// TIA Portal project "Pompe" (V15.1)

(* hardware
DEVICE "S71500/ET200MP station_1"  S7-1500 station
   slot 0: "Rail_0"  Rack  6ES7 590-1***0-0AA0
   slot 1: "PLC_1"  CPU 1513-1 PN  6ES7 513-1AL02-0AB0  V2.6
      slot 3: "CPU display_1"  6ES7591-1AA00-0AA0
DEVICE "HMI_1"  KTP900 Basic PN
   slot 0: "HMI_1"  KTP900 Basic PN  6AV2 123-2JB03-0AX0  15.1.0.0
   slot 1: "HMI_RT_1"  KTP900 Basic PN  6AV2 123-2JB03-0AX0  15.1.0.0
   slot 5: "HMI_1.IE_CP_1"  PROFINET Interface  15.0.1.0
      slot 1: "PROFINET Interface_1"  PROFINET Interface
         slot 1: "Port_1"  Port
*)

// ===== PLC "PLC_1"  CPU 1513-1 PN =====

VAR_GLOBAL   // PLC tag table "Default tag table"
   "Clock_Byte" AT %MB0 : Byte;
   "Clock_10Hz" AT %M0.0 : Bool;
   "Clock_5Hz" AT %M0.1 : Bool;
   "Clock_2.5Hz" AT %M0.2 : Bool;
   "Clock_2Hz" AT %M0.3 : Bool;
   "Clock_1.25Hz" AT %M0.4 : Bool;
   "Clock_1Hz" AT %M0.5 : Bool;
   "Clock_0.625Hz" AT %M0.6 : Bool;
   "Clock_0.5Hz" AT %M0.7 : Bool;
END_VAR

DATA_BLOCK "Pompa_DB"   // DB1
{ S7_Optimized_Access := 'TRUE' }
VERSION : 0.1
   VAR
      comanda_start : Bool;
      comanda_oprire : Bool;
      feedback : Bool;
      pornire_succes : Bool;
   END_VAR
BEGIN
END_DATA_BLOCK

DATA_BLOCK "Bazin_DB"   // DB2
{ S7_Optimized_Access := 'TRUE' }
VERSION : 0.1
   VAR
      volum_maxim : Real := 100.0;
      volum_curent : Real;
      gol : Bool;
      plin : Bool;
   END_VAR
BEGIN
END_DATA_BLOCK

DATA_BLOCK "Robinet_DB"   // DB3
{ S7_Optimized_Access := 'TRUE' }
VERSION : 0.1
   VAR
      comanda_pornire : Bool;
      pornit : Bool;
      comanda_oprire : Bool;
   END_VAR
BEGIN
END_DATA_BLOCK

DATA_BLOCK "Alarme"   // DB4
{ S7_Optimized_Access := 'TRUE' }
VERSION : 0.1
   VAR
      alarme_gather : Word;
      alarme_vect : Array[0..15] of Bool;
   END_VAR
BEGIN
END_DATA_BLOCK

DATA_BLOCK "Avarii"   // DB5
{ S7_Optimized_Access := 'TRUE' }
VERSION : 0.1
   VAR
      esd : Bool;
      btn_esd : Bool;
      btn_reset_esd : Bool;
      avarie_pompa_1 : Bool;
      avarie_pompa_auxiliara : Bool;
      avarie_robinet : Bool;
      avarie_generala : Bool;
      reset_avarie_generala : Bool;
   END_VAR
BEGIN
END_DATA_BLOCK

DATA_BLOCK "Butoane/Permisiuni"   // DB6
{ S7_Optimized_Access := 'TRUE' }
VERSION : 0.1
BEGIN
END_DATA_BLOCK

DATA_BLOCK "Simulare_DB"   // DB9
{ S7_Optimized_Access := 'TRUE' }
VERSION : 0.1
   VAR
      mod_selectat : USInt;
      paritate_mod : USInt;
      pompa_oprita_hmi : Bool;
      pompa_aux_oprita_hmi : Bool;
      robinet_oprit_hmi : Bool;
      nivel_de_mentinut : Real;
   END_VAR
BEGIN
END_DATA_BLOCK

DATA_BLOCK "Bazin_DB_1"   // DB10
{ S7_Optimized_Access := 'TRUE' }
VERSION : 0.1
// stored: InstanceOfName Bazin
"Bazin"
BEGIN
END_DATA_BLOCK

DATA_BLOCK "Robinet_DB_1"   // DB11
{ S7_Optimized_Access := 'TRUE' }
VERSION : 0.1
// stored: InstanceOfName Robinet
"Robinet"
BEGIN
END_DATA_BLOCK

DATA_BLOCK "Auxiliare"   // DB12
{ S7_Optimized_Access := 'TRUE' }
VERSION : 0.1
   VAR
      enable_network : Bool := false;
   END_VAR
BEGIN
END_DATA_BLOCK

DATA_BLOCK "Vana_DB"   // DB13
{ S7_Optimized_Access := 'TRUE' }
VERSION : 0.1
   VAR
      comanda_start : Bool;
      comanda_oprire : Bool;
      feedback : Bool;
      pornire_succes : Bool;
   END_VAR
BEGIN
END_DATA_BLOCK

DATA_BLOCK "Vana_DB_1"   // DB14
{ S7_Optimized_Access := 'TRUE' }
VERSION : 0.1
// stored: InstanceOfName Vana
"Vana"
BEGIN
END_DATA_BLOCK

DATA_BLOCK "Pompa_DB_1"   // DB15
{ S7_Optimized_Access := 'TRUE' }
VERSION : 0.1
// stored: InstanceOfName Pompa
"Pompa"
BEGIN
END_DATA_BLOCK

DATA_BLOCK "Simulare_DB_1"   // DB16
{ S7_Optimized_Access := 'TRUE' }
VERSION : 0.1
// stored: InstanceOfName Simulare
"Simulare"
BEGIN
END_DATA_BLOCK

DATA_BLOCK "Pompa_DB_2"   // DB17
{ S7_Optimized_Access := 'TRUE' }
VERSION : 0.1
// stored: InstanceOfName Pompa
"Pompa"
BEGIN
END_DATA_BLOCK

DATA_BLOCK "Pompa_auxiliara_DB"   // DB18
{ S7_Optimized_Access := 'TRUE' }
VERSION : 0.1
   VAR
      comanda_start : Bool;
      comanda_oprire : Bool;
      feedback : Bool;
      pornire_succes : Bool;
      btn_pornire : Bool;
   END_VAR
BEGIN
END_DATA_BLOCK

// folder: System blocks/Program resources

DATA_BLOCK "Timer_reset_ESD"   // DB7
{ S7_Optimized_Access := 'TRUE' }
AUTHOR : Simatic
FAMILY : IEC
NAME : IEC_TMR
VERSION : 1.0
// stored: InstanceOfName IEC_TIMER
"IEC_TIMER"
BEGIN
END_DATA_BLOCK

DATA_BLOCK "Timer_reset_avarie_generala"   // DB8
{ S7_Optimized_Access := 'TRUE' }
AUTHOR : Simatic
FAMILY : IEC
NAME : IEC_TMR
VERSION : 1.0
// stored: InstanceOfName IEC_TIMER
"IEC_TIMER"
BEGIN
END_DATA_BLOCK

// folder: (top level)

FUNCTION_BLOCK "Pompa"   // FB1, LAD
{ S7_Optimized_Access := 'TRUE' }
VERSION : 0.1
   VAR_INPUT
      esd : Bool;
      avarie : Bool;
      mod_selectat : USInt;
      comanda_oprire : Bool;
   END_VAR
   VAR_OUTPUT
      feedback : Bool;
      pornire_succes : Bool;
   END_VAR
   VAR_IN_OUT
      comanda_start : Bool;
   END_VAR
   VAR
      pornire : Bool;
      timer_confirmare : TON_TIME;
   END_VAR
BEGIN

REGION Network 1: Comanda plecare
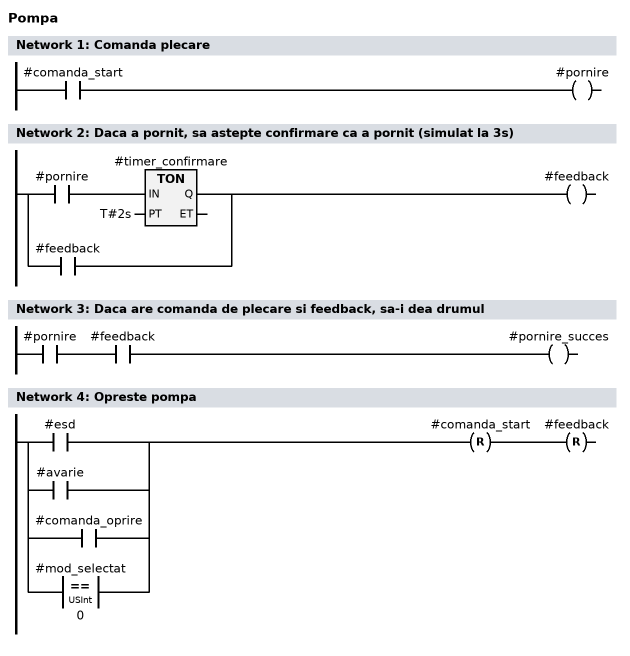
   RUNG wire#powerrail
      Contact( #comanda_start )
      Coil( #pornire )
   END_RUNG
   // the same network as SCL:
   #pornire := #comanda_start;
END_REGION

REGION Network 2: Daca a pornit, sa astepte confirmare ca a pornit (simulat la 3s)
   #timer_confirmare(IN := #pornire, PT := T#2s);   // TON
   #feedback := #timer_confirmare.Q OR #feedback;
END_REGION

REGION Network 3: Daca are comanda de plecare si feedback, sa-i dea drumul
   RUNG wire#powerrail
      Contact( #pornire )
      Contact( #feedback )
      Coil( #pornire_succes )
   END_RUNG
   // the same network as SCL:
   #pornire_succes := #pornire AND #feedback;
END_REGION

REGION Network 4: Opreste pompa
   RUNG wire#powerrail
      Contact( #esd )
      wire#w1
      R_Coil( #comanda_start )
      R_Coil( #feedback )
   END_RUNG
   RUNG wire#powerrail
      Contact( #avarie )
   END_RUNG wire#w1
   RUNG wire#powerrail
      Contact( #comanda_oprire )
   END_RUNG wire#w1
   RUNG wire#powerrail
      { S7_Templates := "SrcType := USInt" } EQ_Contact(in1 := #mod_selectat, in2 := 0)
   END_RUNG wire#w1
   // the same network as SCL:
   IF #esd OR #avarie OR #comanda_oprire OR (#mod_selectat = 0) THEN
       #comanda_start := FALSE;
       #feedback := FALSE;
   END_IF;
END_REGION
END_FUNCTION_BLOCK

FUNCTION_BLOCK "Bazin"   // FB2, LAD
{ S7_Optimized_Access := 'TRUE' }
VERSION : 0.1
   VAR_INPUT
      volum_maxim : Real;
   END_VAR
   VAR_OUTPUT
      gol : Bool;
      plin : Bool;
   END_VAR
   VAR_IN_OUT
      volum_curent : Real;
   END_VAR
BEGIN

REGION Network 1: Setare gol
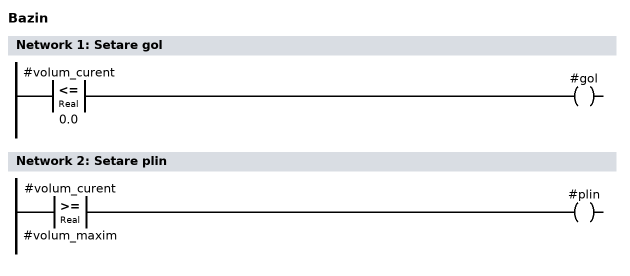
   RUNG wire#powerrail
      { S7_Templates := "SrcType := Real" } LE_Contact(in1 := #volum_curent, in2 := 0.0)
      Coil( #gol )
   END_RUNG
   // the same network as SCL:
   #gol := #volum_curent <= 0.0;
END_REGION

REGION Network 2: Setare plin
   RUNG wire#powerrail
      { S7_Templates := "SrcType := Real" } GE_Contact(in1 := #volum_curent, in2 := #volum_maxim)
      Coil( #plin )
   END_RUNG
   // the same network as SCL:
   #plin := #volum_curent >= #volum_maxim;
END_REGION
END_FUNCTION_BLOCK

FUNCTION_BLOCK "Robinet"   // FB3, LAD
{ S7_Optimized_Access := 'TRUE' }
VERSION : 0.1
   VAR_INPUT
      esd : Bool;
      avarie : Bool;
      comanda_oprire : Bool;
   END_VAR
   VAR_IN_OUT
      pornit : Bool;
      btn_pornire : Bool;
   END_VAR
BEGIN

REGION Network 1: Sa aiba permisiunea de pornire
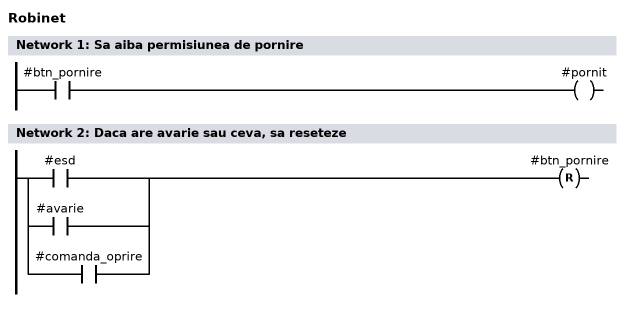
   RUNG wire#powerrail
      Contact( #btn_pornire )
      Coil( #pornit )
   END_RUNG
   // the same network as SCL:
   #pornit := #btn_pornire;
END_REGION

REGION Network 2: Daca are avarie sau ceva, sa reseteze
   RUNG wire#powerrail
      Contact( #esd )
      wire#w1
      R_Coil( #btn_pornire )
   END_RUNG
   RUNG wire#powerrail
      Contact( #avarie )
   END_RUNG wire#w1
   RUNG wire#powerrail
      Contact( #comanda_oprire )
   END_RUNG wire#w1
   // the same network as SCL:
   IF #esd OR #avarie OR #comanda_oprire THEN #btn_pornire := FALSE; END_IF;
END_REGION
END_FUNCTION_BLOCK

FUNCTION_BLOCK "Simulare"   // FB4, LAD
{ S7_Optimized_Access := 'TRUE' }
VERSION : 0.1
   VAR_INPUT
      plin : Bool;
      gol : Bool;
      pompa_pornita : Bool;
      pompa_aux_pornita : Bool;
      robinet_pornit : Bool;
      esd : Bool;
      avarie_pompa : Bool;
      avarie_pompa_aux : Bool;
      avarie_robinet : Bool;
      nivel_de_mentinut : Real;
   END_VAR
   VAR_OUTPUT
      start_pompa : Bool;
      start_pompa_aux : Bool;
      start_robinet : Bool;
      opreste_pompa : Bool;
      opreste_pompa_aux : Bool;
      opreste_robinet : Bool;
      pompa_oprita_hmi : Bool;
      pompa_oprita_aux_hmi : Bool;
      robinet_oprit_hmi : Bool;
   END_VAR
   VAR_IN_OUT
      btn_pompa_aux : Bool;
      volum_curent : Real;
      mod_functionare : USInt;
   END_VAR
   VAR
      re1 : Bool;
      re2 : Bool;
      re3 : Bool;
      lim_inf : Real;
      lim_sup : Real;
   END_VAR
   VAR_TEMP   // added for the SCL form of the ladder/FBD networks
      _w1 : Bool;
      _w2 : Bool;
   END_VAR
BEGIN

REGION Network 1: Calcul limite noi
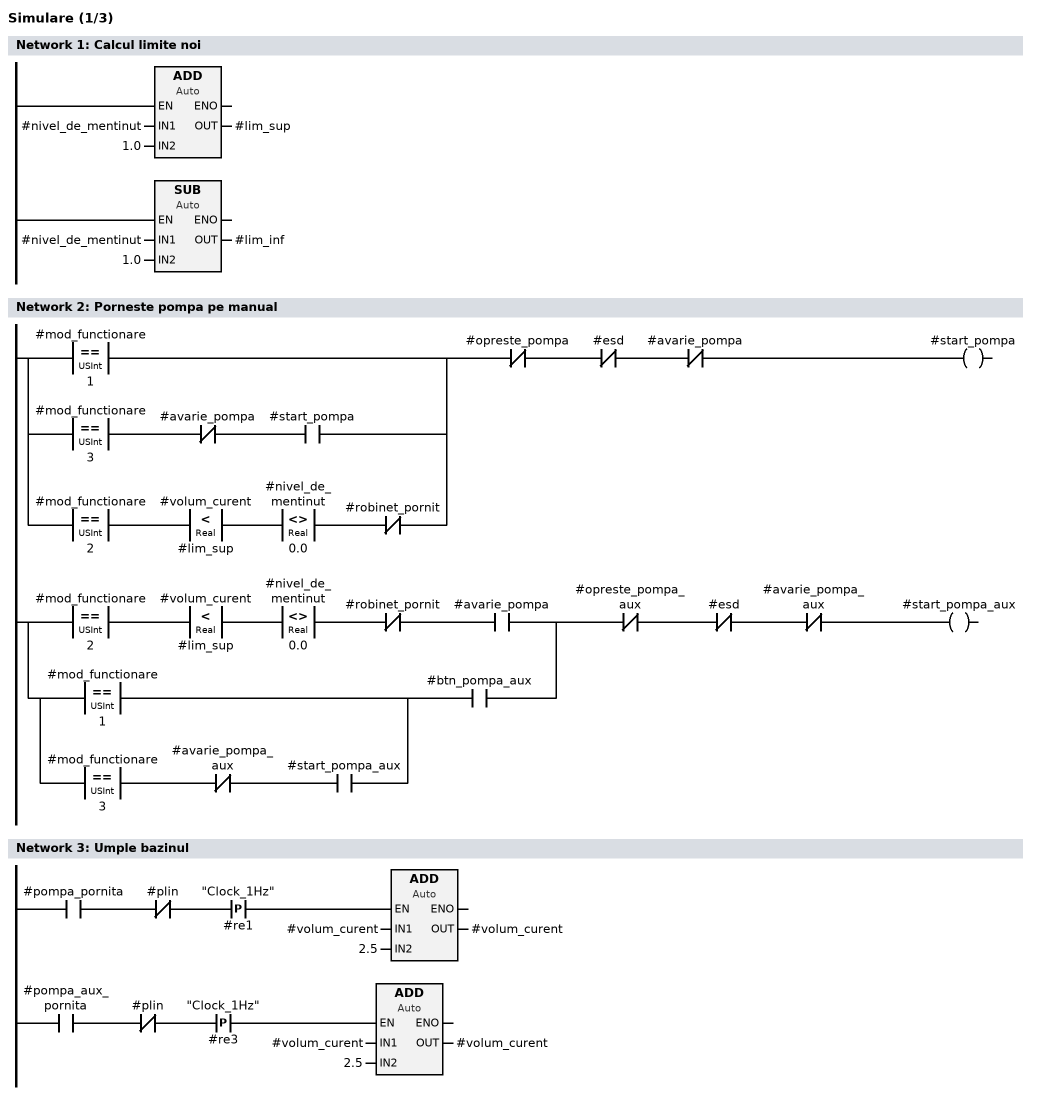
   RUNG wire#powerrail
      Add(in1 := #nivel_de_mentinut, in2 := 1.0, out => #lim_sup)
   END_RUNG
   RUNG wire#powerrail
      Sub(in1 := #nivel_de_mentinut, in2 := 1.0, out => #lim_inf)
   END_RUNG
   // the same network as SCL:
   #lim_sup := #nivel_de_mentinut + 1.0;
   #lim_inf := #nivel_de_mentinut - 1.0;
END_REGION

REGION Network 2: Porneste pompa pe manual
   RUNG wire#powerrail
      { S7_Templates := "SrcType := USInt" } EQ_Contact(in1 := #mod_functionare, in2 := 1)
      wire#w1
      I_Contact( #opreste_pompa )
      I_Contact( #esd )
      I_Contact( #avarie_pompa )
      Coil( #start_pompa )
   END_RUNG
   RUNG wire#powerrail
      { S7_Templates := "SrcType := USInt" } EQ_Contact(in1 := #mod_functionare, in2 := 3)
      I_Contact( #avarie_pompa )
      Contact( #start_pompa )
   END_RUNG wire#w1
   RUNG wire#powerrail
      { S7_Templates := "SrcType := USInt" } EQ_Contact(in1 := #mod_functionare, in2 := 2)
      { S7_Templates := "SrcType := Real" } LT_Contact(in1 := #volum_curent, in2 := #lim_sup)
      { S7_Templates := "SrcType := Real" } NE_Contact(in1 := #nivel_de_mentinut, in2 := 0.0)
      I_Contact( #robinet_pornit )
   END_RUNG wire#w1
   RUNG wire#powerrail
      { S7_Templates := "SrcType := USInt" } EQ_Contact(in1 := #mod_functionare, in2 := 2)
      { S7_Templates := "SrcType := Real" } LT_Contact(in1 := #volum_curent, in2 := #lim_sup)
      { S7_Templates := "SrcType := Real" } NE_Contact(in1 := #nivel_de_mentinut, in2 := 0.0)
      I_Contact( #robinet_pornit )
      Contact( #avarie_pompa )
      wire#w2
      I_Contact( #opreste_pompa_aux )
      I_Contact( #esd )
      I_Contact( #avarie_pompa_aux )
      Coil( #start_pompa_aux )
   END_RUNG
   RUNG wire#powerrail
      { S7_Templates := "SrcType := USInt" } EQ_Contact(in1 := #mod_functionare, in2 := 1)
      wire#w3
      Contact( #btn_pompa_aux )
   END_RUNG wire#w2
   RUNG wire#powerrail
      { S7_Templates := "SrcType := USInt" } EQ_Contact(in1 := #mod_functionare, in2 := 3)
      I_Contact( #avarie_pompa_aux )
      Contact( #start_pompa_aux )
   END_RUNG wire#w3
   // the same network as SCL:
   #start_pompa := ((#mod_functionare = 1) OR ((#mod_functionare = 3) AND NOT #avarie_pompa AND #start_pompa) OR ((#mod_functionare = 2) AND (#volum_curent < #lim_sup) AND (#nivel_de_mentinut <> 0.0) AND NOT #robinet_pornit)) AND NOT #opreste_pompa AND NOT #esd AND NOT #avarie_pompa;
   #start_pompa_aux := (((#mod_functionare = 2) AND (#volum_curent < #lim_sup) AND (#nivel_de_mentinut <> 0.0) AND NOT #robinet_pornit AND #avarie_pompa) OR (((#mod_functionare = 1) OR ((#mod_functionare = 3) AND NOT #avarie_pompa_aux AND #start_pompa_aux)) AND #btn_pompa_aux)) AND NOT #opreste_pompa_aux AND NOT #esd AND NOT #avarie_pompa_aux;
END_REGION

REGION Network 3: Umple bazinul
   RUNG wire#powerrail
      Contact( #pompa_pornita )
      I_Contact( #plin )
      P_Contact(operand := "Clock_1Hz", bit := #re1)
      Add(in1 := #volum_curent, in2 := 2.5, out => #volum_curent)
   END_RUNG
   RUNG wire#powerrail
      Contact( #pompa_aux_pornita )
      I_Contact( #plin )
      P_Contact(operand := "Clock_1Hz", bit := #re3)
      Add(in1 := #volum_curent, in2 := 2.5, out => #volum_curent)
   END_RUNG
   // the same network as SCL:
   #_w1 := #pompa_pornita AND NOT #plin AND "Clock_1Hz" AND NOT #re1;   // rising edge of "Clock_1Hz"
   #re1 := "Clock_1Hz";
   IF #_w1 THEN #volum_curent := #volum_curent + 2.5; END_IF;
   #_w2 := #pompa_aux_pornita AND NOT #plin AND "Clock_1Hz" AND NOT #re3;   // rising edge of "Clock_1Hz"
   #re3 := "Clock_1Hz";
   IF #_w2 THEN #volum_curent := #volum_curent + 2.5; END_IF;
END_REGION

REGION Network 4: Opreste pompa/pompa aux
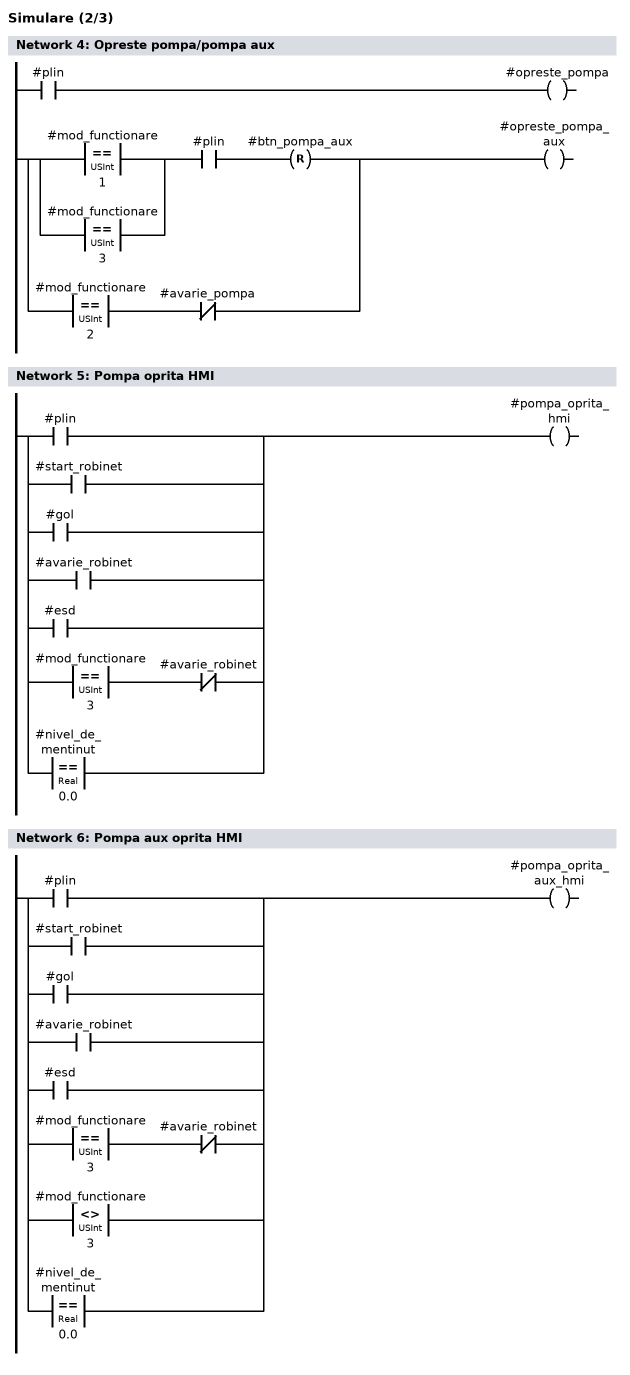
   RUNG wire#powerrail
      Contact( #plin )
      Coil( #opreste_pompa )
   END_RUNG
   RUNG wire#powerrail
      { S7_Templates := "SrcType := USInt" } EQ_Contact(in1 := #mod_functionare, in2 := 1)
      wire#w1
      Contact( #plin )
      R_Coil( #btn_pompa_aux )
      wire#w2
      Coil( #opreste_pompa_aux )
   END_RUNG
   RUNG wire#powerrail
      { S7_Templates := "SrcType := USInt" } EQ_Contact(in1 := #mod_functionare, in2 := 3)
   END_RUNG wire#w1
   RUNG wire#powerrail
      { S7_Templates := "SrcType := USInt" } EQ_Contact(in1 := #mod_functionare, in2 := 2)
      I_Contact( #avarie_pompa )
   END_RUNG wire#w2
   // the same network as SCL:
   #opreste_pompa := #plin;
   #_w1 := ((#mod_functionare = 1) OR (#mod_functionare = 3)) AND #plin;
   IF #_w1 THEN #btn_pompa_aux := FALSE; END_IF;
   #opreste_pompa_aux := #_w1 OR ((#mod_functionare = 2) AND NOT #avarie_pompa);
END_REGION

REGION Network 5: Pompa oprita HMI
   RUNG wire#powerrail
      Contact( #plin )
      wire#w1
      Coil( #pompa_oprita_hmi )
   END_RUNG
   RUNG wire#powerrail
      Contact( #start_robinet )
   END_RUNG wire#w1
   RUNG wire#powerrail
      Contact( #gol )
   END_RUNG wire#w1
   RUNG wire#powerrail
      Contact( #avarie_robinet )
   END_RUNG wire#w1
   RUNG wire#powerrail
      Contact( #esd )
   END_RUNG wire#w1
   RUNG wire#powerrail
      { S7_Templates := "SrcType := USInt" } EQ_Contact(in1 := #mod_functionare, in2 := 3)
      I_Contact( #avarie_robinet )
   END_RUNG wire#w1
   RUNG wire#powerrail
      { S7_Templates := "SrcType := Real" } EQ_Contact(in1 := #nivel_de_mentinut, in2 := 0.0)
   END_RUNG wire#w1
   // the same network as SCL:
   #pompa_oprita_hmi := #plin OR #start_robinet OR #gol OR #avarie_robinet OR #esd OR ((#mod_functionare = 3) AND NOT #avarie_robinet) OR (#nivel_de_mentinut = 0.0);
END_REGION

REGION Network 6: Pompa aux oprita HMI
   RUNG wire#powerrail
      Contact( #plin )
      wire#w1
      Coil( #pompa_oprita_aux_hmi )
   END_RUNG
   RUNG wire#powerrail
      Contact( #start_robinet )
   END_RUNG wire#w1
   RUNG wire#powerrail
      Contact( #gol )
   END_RUNG wire#w1
   RUNG wire#powerrail
      Contact( #avarie_robinet )
   END_RUNG wire#w1
   RUNG wire#powerrail
      Contact( #esd )
   END_RUNG wire#w1
   RUNG wire#powerrail
      { S7_Templates := "SrcType := USInt" } EQ_Contact(in1 := #mod_functionare, in2 := 3)
      I_Contact( #avarie_robinet )
   END_RUNG wire#w1
   RUNG wire#powerrail
      { S7_Templates := "SrcType := USInt" } NE_Contact(in1 := #mod_functionare, in2 := 3)
   END_RUNG wire#w1
   RUNG wire#powerrail
      { S7_Templates := "SrcType := Real" } EQ_Contact(in1 := #nivel_de_mentinut, in2 := 0.0)
   END_RUNG wire#w1
   // the same network as SCL:
   #pompa_oprita_aux_hmi := #plin OR #start_robinet OR #gol OR #avarie_robinet OR #esd OR ((#mod_functionare = 3) AND NOT #avarie_robinet) OR (#mod_functionare <> 3) OR (#nivel_de_mentinut = 0.0);
END_REGION

REGION Network 7: Robinet oprit HMI
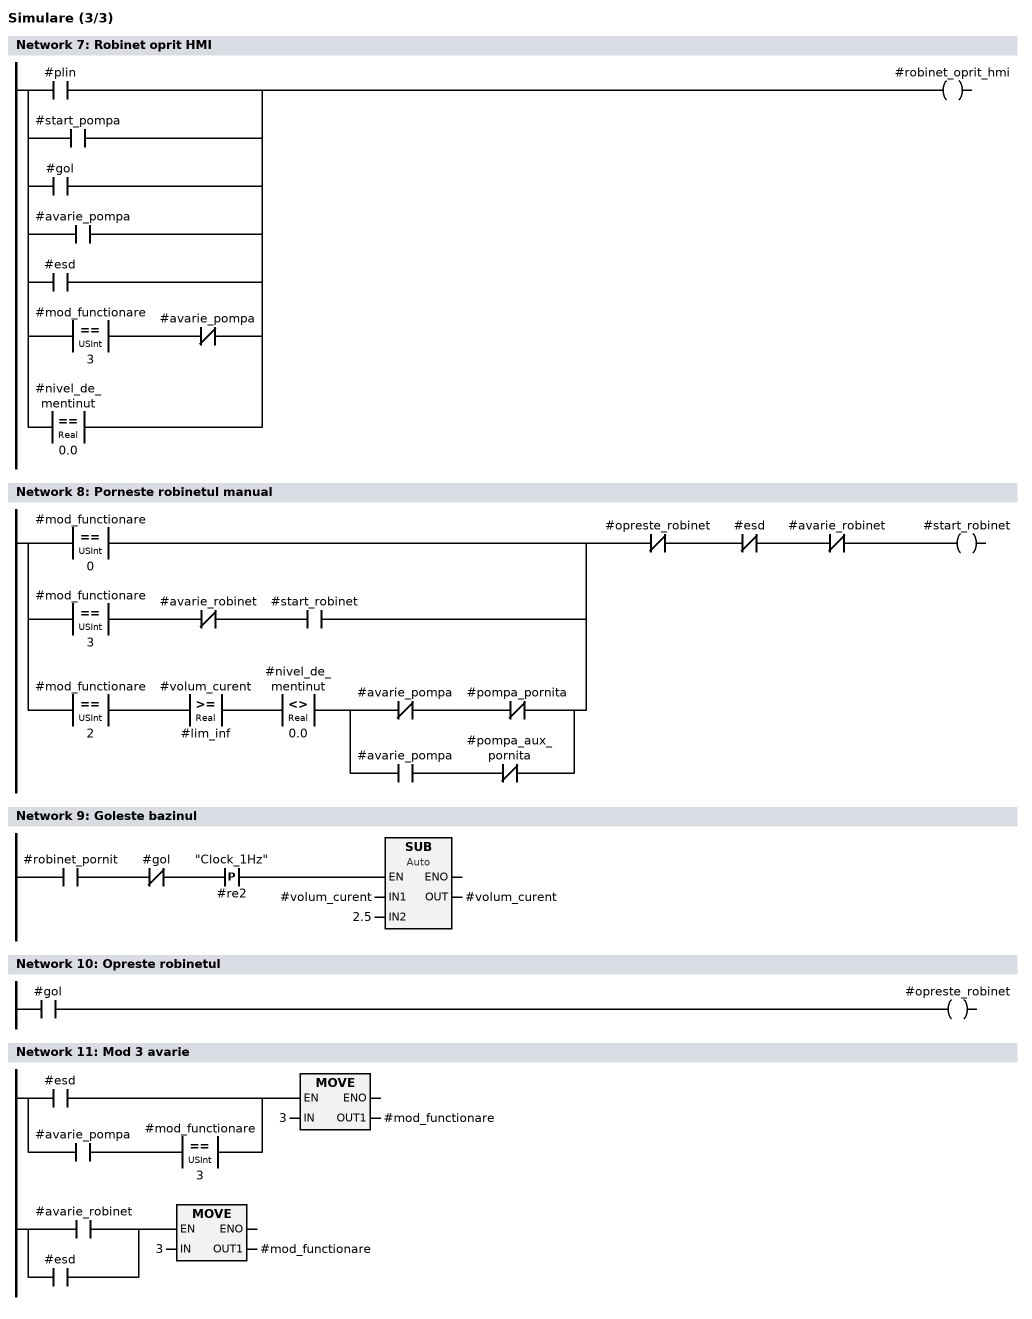
   RUNG wire#powerrail
      Contact( #plin )
      wire#w1
      Coil( #robinet_oprit_hmi )
   END_RUNG
   RUNG wire#powerrail
      Contact( #start_pompa )
   END_RUNG wire#w1
   RUNG wire#powerrail
      Contact( #gol )
   END_RUNG wire#w1
   RUNG wire#powerrail
      Contact( #avarie_pompa )
   END_RUNG wire#w1
   RUNG wire#powerrail
      Contact( #esd )
   END_RUNG wire#w1
   RUNG wire#powerrail
      { S7_Templates := "SrcType := USInt" } EQ_Contact(in1 := #mod_functionare, in2 := 3)
      I_Contact( #avarie_pompa )
   END_RUNG wire#w1
   RUNG wire#powerrail
      { S7_Templates := "SrcType := Real" } EQ_Contact(in1 := #nivel_de_mentinut, in2 := 0.0)
   END_RUNG wire#w1
   // the same network as SCL:
   #robinet_oprit_hmi := #plin OR #start_pompa OR #gol OR #avarie_pompa OR #esd OR ((#mod_functionare = 3) AND NOT #avarie_pompa) OR (#nivel_de_mentinut = 0.0);
END_REGION

REGION Network 8: Porneste robinetul manual
   RUNG wire#powerrail
      { S7_Templates := "SrcType := USInt" } EQ_Contact(in1 := #mod_functionare, in2 := 0)
      wire#w1
      I_Contact( #opreste_robinet )
      I_Contact( #esd )
      I_Contact( #avarie_robinet )
      Coil( #start_robinet )
   END_RUNG
   RUNG wire#powerrail
      { S7_Templates := "SrcType := USInt" } EQ_Contact(in1 := #mod_functionare, in2 := 3)
      I_Contact( #avarie_robinet )
      Contact( #start_robinet )
   END_RUNG wire#w1
   RUNG wire#powerrail
      { S7_Templates := "SrcType := USInt" } EQ_Contact(in1 := #mod_functionare, in2 := 2)
      { S7_Templates := "SrcType := Real" } GE_Contact(in1 := #volum_curent, in2 := #lim_inf)
      { S7_Templates := "SrcType := Real" } NE_Contact(in1 := #nivel_de_mentinut, in2 := 0.0)
      wire#w2
      I_Contact( #avarie_pompa )
      I_Contact( #pompa_pornita )
   END_RUNG wire#w1
   RUNG wire#w2
      Contact( #avarie_pompa )
      I_Contact( #pompa_aux_pornita )
   END_RUNG wire#w1
   // the same network as SCL:
   #start_robinet := ((#mod_functionare = 0) OR ((#mod_functionare = 3) AND NOT #avarie_robinet AND #start_robinet) OR ((#mod_functionare = 2) AND (#volum_curent >= #lim_inf) AND (#nivel_de_mentinut <> 0.0) AND ((NOT #avarie_pompa AND NOT #pompa_pornita) OR (#avarie_pompa AND NOT #pompa_aux_pornita)))) AND NOT #opreste_robinet AND NOT #esd AND NOT #avarie_robinet;
END_REGION

REGION Network 9: Goleste bazinul
   RUNG wire#powerrail
      Contact( #robinet_pornit )
      I_Contact( #gol )
      P_Contact(operand := "Clock_1Hz", bit := #re2)
      Sub(in1 := #volum_curent, in2 := 2.5, out => #volum_curent)
   END_RUNG
   // the same network as SCL:
   #_w1 := #robinet_pornit AND NOT #gol AND "Clock_1Hz" AND NOT #re2;   // rising edge of "Clock_1Hz"
   #re2 := "Clock_1Hz";
   IF #_w1 THEN #volum_curent := #volum_curent - 2.5; END_IF;
END_REGION

REGION Network 10: Opreste robinetul
   RUNG wire#powerrail
      Contact( #gol )
      Coil( #opreste_robinet )
   END_RUNG
   // the same network as SCL:
   #opreste_robinet := #gol;
END_REGION

REGION Network 11: Mod 3 avarie
   RUNG wire#powerrail
      Contact( #esd )
      wire#w1
      Move(in := 3, out1 => #mod_functionare)
   END_RUNG
   RUNG wire#powerrail
      Contact( #avarie_pompa )
      { S7_Templates := "SrcType := USInt" } EQ_Contact(in1 := #mod_functionare, in2 := 3)
   END_RUNG wire#w1
   RUNG wire#powerrail
      Contact( #avarie_robinet )
      wire#w2
      Move(in := 3, out1 => #mod_functionare)
   END_RUNG
   RUNG wire#powerrail
      Contact( #esd )
   END_RUNG wire#w2
   // the same network as SCL:
   IF #esd OR (#avarie_pompa AND (#mod_functionare = 3)) THEN #mod_functionare := 3; END_IF;
   IF #avarie_robinet OR #esd THEN #mod_functionare := 3; END_IF;
END_REGION
END_FUNCTION_BLOCK

FUNCTION_BLOCK "Vana"   // FB5, LAD
{ S7_Optimized_Access := 'TRUE' }
VERSION : 0.1
   VAR_INPUT
      esd : Bool;
      avarie : Bool;
      comanda_oprire : Bool;
      mod_selectat : USInt;
   END_VAR
   VAR_OUTPUT
      feedback : Bool;
      pornire_succes : Bool;
   END_VAR
   VAR_IN_OUT
      comanda_start : Bool;
   END_VAR
   VAR
      pornire : Bool;
      timer_confirmare : TON_TIME;
   END_VAR
BEGIN

REGION Network 1: Comanda plecare
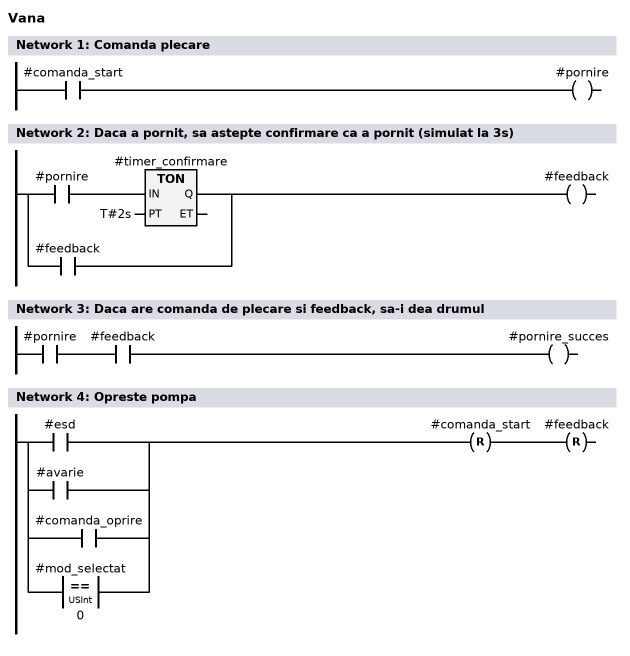
   RUNG wire#powerrail
      Contact( #comanda_start )
      Coil( #pornire )
   END_RUNG
   // the same network as SCL:
   #pornire := #comanda_start;
END_REGION

REGION Network 2: Daca a pornit, sa astepte confirmare ca a pornit (simulat la 3s)
   #timer_confirmare(IN := #pornire, PT := T#2s);   // TON
   #feedback := #timer_confirmare.Q OR #feedback;
END_REGION

REGION Network 3: Daca are comanda de plecare si feedback, sa-i dea drumul
   RUNG wire#powerrail
      Contact( #pornire )
      Contact( #feedback )
      Coil( #pornire_succes )
   END_RUNG
   // the same network as SCL:
   #pornire_succes := #pornire AND #feedback;
END_REGION

REGION Network 4: Opreste pompa
   RUNG wire#powerrail
      Contact( #esd )
      wire#w1
      R_Coil( #comanda_start )
      R_Coil( #feedback )
   END_RUNG
   RUNG wire#powerrail
      Contact( #avarie )
   END_RUNG wire#w1
   RUNG wire#powerrail
      Contact( #comanda_oprire )
   END_RUNG wire#w1
   RUNG wire#powerrail
      { S7_Templates := "SrcType := USInt" } EQ_Contact(in1 := #mod_selectat, in2 := 0)
   END_RUNG wire#w1
   // the same network as SCL:
   IF #esd OR #avarie OR #comanda_oprire OR (#mod_selectat = 0) THEN
       #comanda_start := FALSE;
       #feedback := FALSE;
   END_IF;
END_REGION
END_FUNCTION_BLOCK

ORGANIZATION_BLOCK "Main"   // OB1, LAD, ProgramCycle
TITLE = "Main Program Sweep (Cycle)"
{ S7_Optimized_Access := 'TRUE' }
VERSION : 0.1
   VAR_INPUT
      Initial_Call : Bool;   // Initial call of this OB
      Remanence : Bool;   // =True, if remanent data are available
   END_VAR
BEGIN

REGION Network 1: Gather de alarme
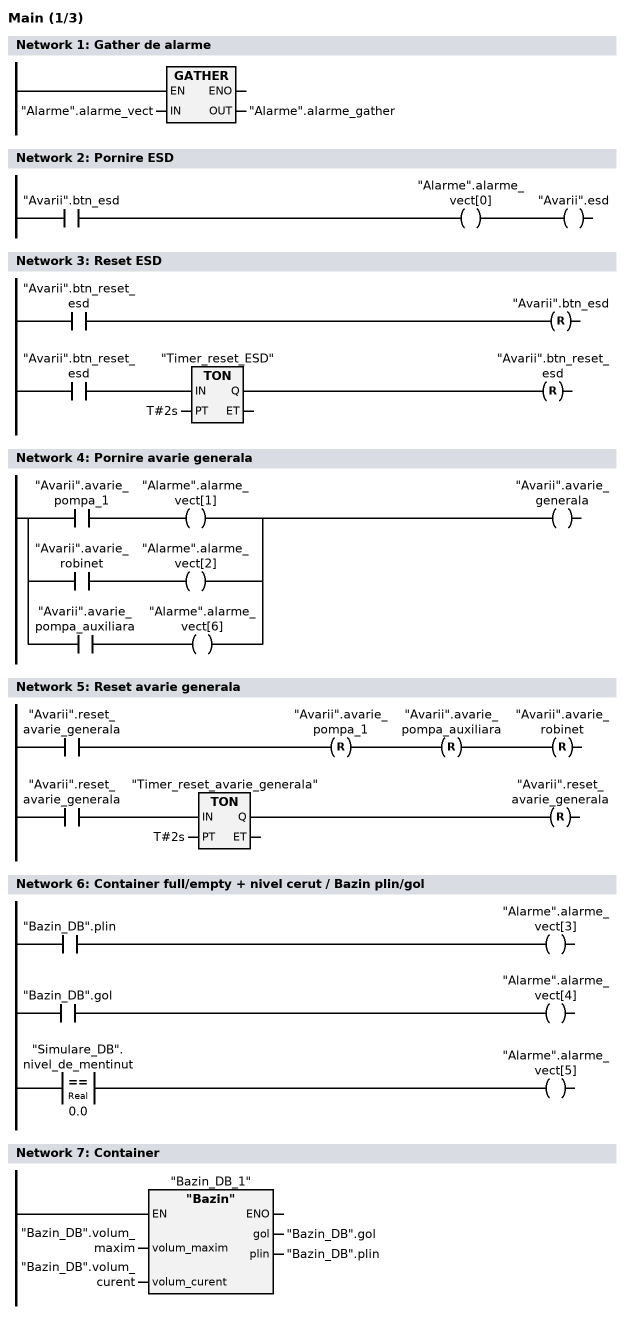
   GATHER(IN := "Alarme".alarme_vect, OUT => "Alarme".alarme_gather);
END_REGION

REGION Network 2: Pornire ESD
   RUNG wire#powerrail
      Contact( "Avarii".btn_esd )
      Coil( "Alarme".alarme_vect[0] )
      Coil( "Avarii".esd )
   END_RUNG
   // the same network as SCL:
   "Alarme".alarme_vect[0] := "Avarii".btn_esd;
   "Avarii".esd := "Avarii".btn_esd;
END_REGION

REGION Network 3: Reset ESD
   IF "Avarii".btn_reset_esd THEN "Avarii".btn_esd := FALSE; END_IF;
   "Timer_reset_ESD".TON(IN := "Avarii".btn_reset_esd, PT := T#2s);
   IF "Timer_reset_ESD".Q THEN "Avarii".btn_reset_esd := FALSE; END_IF;
END_REGION

REGION Network 4: Pornire avarie generala
   RUNG wire#powerrail
      Contact( "Avarii".avarie_pompa_1 )
      Coil( "Alarme".alarme_vect[1] )
      wire#w1
      Coil( "Avarii".avarie_generala )
   END_RUNG
   RUNG wire#powerrail
      Contact( "Avarii".avarie_robinet )
      Coil( "Alarme".alarme_vect[2] )
   END_RUNG wire#w1
   RUNG wire#powerrail
      Contact( "Avarii".avarie_pompa_auxiliara )
      Coil( "Alarme".alarme_vect[6] )
   END_RUNG wire#w1
   // the same network as SCL:
   "Alarme".alarme_vect[1] := "Avarii".avarie_pompa_1;
   "Alarme".alarme_vect[2] := "Avarii".avarie_robinet;
   "Alarme".alarme_vect[6] := "Avarii".avarie_pompa_auxiliara;
   "Avarii".avarie_generala := "Avarii".avarie_pompa_1 OR "Avarii".avarie_robinet OR "Avarii".avarie_pompa_auxiliara;
END_REGION

REGION Network 5: Reset avarie generala
   IF "Avarii".reset_avarie_generala THEN
       "Avarii".avarie_pompa_1 := FALSE;
       "Avarii".avarie_pompa_auxiliara := FALSE;
       "Avarii".avarie_robinet := FALSE;
   END_IF;
   "Timer_reset_avarie_generala".TON(IN := "Avarii".reset_avarie_generala, PT := T#2s);
   IF "Timer_reset_avarie_generala".Q THEN "Avarii".reset_avarie_generala := FALSE; END_IF;
END_REGION

REGION Network 6: Container full/empty + nivel cerut / Bazin plin/gol
   RUNG wire#powerrail
      Contact( "Bazin_DB".plin )
      Coil( "Alarme".alarme_vect[3] )
   END_RUNG
   RUNG wire#powerrail
      Contact( "Bazin_DB".gol )
      Coil( "Alarme".alarme_vect[4] )
   END_RUNG
   RUNG wire#powerrail
      { S7_Templates := "SrcType := Real" } EQ_Contact(in1 := "Simulare_DB".nivel_de_mentinut, in2 := 0.0)
      Coil( "Alarme".alarme_vect[5] )
   END_RUNG
   // the same network as SCL:
   "Alarme".alarme_vect[3] := "Bazin_DB".plin;
   "Alarme".alarme_vect[4] := "Bazin_DB".gol;
   "Alarme".alarme_vect[5] := "Simulare_DB".nivel_de_mentinut = 0.0;
END_REGION

REGION Network 7: Container
   RUNG wire#powerrail
      "Bazin_DB_1"(volum_maxim := "Bazin_DB".volum_maxim, volum_curent := "Bazin_DB".volum_curent, gol => "Bazin_DB".gol, plin => "Bazin_DB".plin)
   END_RUNG
   // the same network as SCL:
   "Bazin_DB_1"(volum_maxim := "Bazin_DB".volum_maxim,   // "Bazin"
                volum_curent := "Bazin_DB".volum_curent,
                gol => "Bazin_DB".gol,
                plin => "Bazin_DB".plin);
END_REGION

REGION Network 8: Robinet
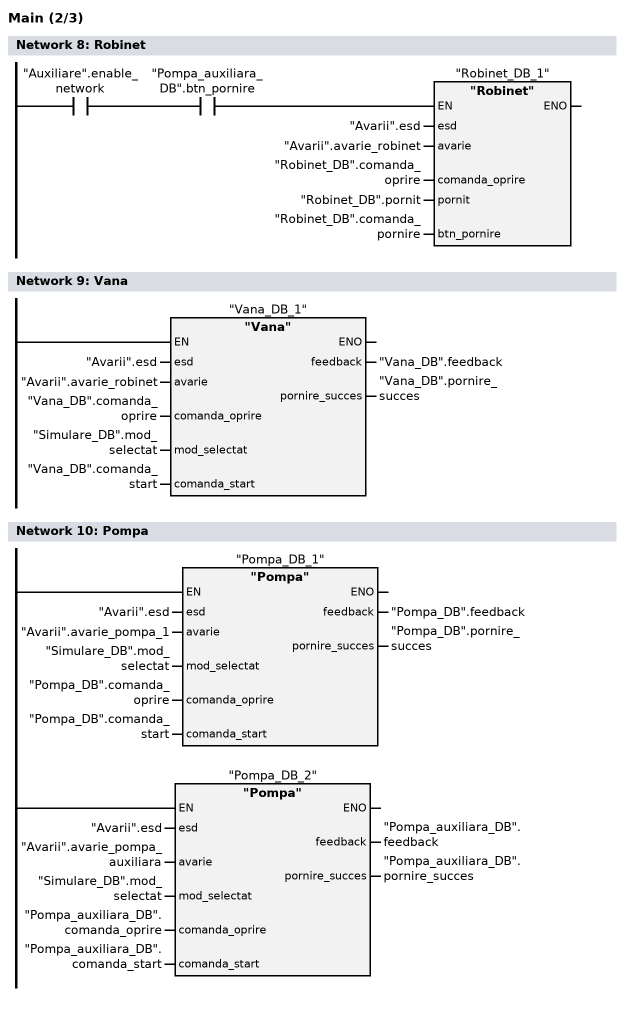
   RUNG wire#powerrail
      Contact( "Auxiliare".enable_network )
      Contact( "Pompa_auxiliara_DB".btn_pornire )
      "Robinet_DB_1"(esd := "Avarii".esd, avarie := "Avarii".avarie_robinet, comanda_oprire := "Robinet_DB".comanda_oprire, pornit := "Robinet_DB".pornit, btn_pornire := "Robinet_DB".comanda_pornire)
   END_RUNG
   // the same network as SCL:
   IF "Auxiliare".enable_network AND "Pompa_auxiliara_DB".btn_pornire THEN
       "Robinet_DB_1"(esd := "Avarii".esd,   // "Robinet"
                      avarie := "Avarii".avarie_robinet,
                      comanda_oprire := "Robinet_DB".comanda_oprire,
                      pornit := "Robinet_DB".pornit,
                      btn_pornire := "Robinet_DB".comanda_pornire);
   END_IF;
END_REGION

REGION Network 9: Vana
   RUNG wire#powerrail
      "Vana_DB_1"(esd := "Avarii".esd, avarie := "Avarii".avarie_robinet, comanda_oprire := "Vana_DB".comanda_oprire, mod_selectat := "Simulare_DB".mod_selectat, comanda_start := "Vana_DB".comanda_start, feedback => "Vana_DB".feedback, pornire_succes => "Vana_DB".pornire_succes)
   END_RUNG
   // the same network as SCL:
   "Vana_DB_1"(esd := "Avarii".esd,   // "Vana"
               avarie := "Avarii".avarie_robinet,
               comanda_oprire := "Vana_DB".comanda_oprire,
               mod_selectat := "Simulare_DB".mod_selectat,
               comanda_start := "Vana_DB".comanda_start,
               feedback => "Vana_DB".feedback,
               pornire_succes => "Vana_DB".pornire_succes);
END_REGION

REGION Network 10: Pompa
   RUNG wire#powerrail
      "Pompa_DB_1"(esd := "Avarii".esd, avarie := "Avarii".avarie_pompa_1, mod_selectat := "Simulare_DB".mod_selectat, comanda_oprire := "Pompa_DB".comanda_oprire, comanda_start := "Pompa_DB".comanda_start, feedback => "Pompa_DB".feedback, pornire_succes => "Pompa_DB".pornire_succes)
   END_RUNG
   RUNG wire#powerrail
      "Pompa_DB_2"(esd := "Avarii".esd, avarie := "Avarii".avarie_pompa_auxiliara, mod_selectat := "Simulare_DB".mod_selectat, comanda_oprire := "Pompa_auxiliara_DB".comanda_oprire, comanda_start := "Pompa_auxiliara_DB".comanda_start, feedback => "Pompa_auxiliara_DB".feedback, pornire_succes => "Pompa_auxiliara_DB".pornire_succes)
   END_RUNG
   // the same network as SCL:
   "Pompa_DB_1"(esd := "Avarii".esd,   // "Pompa"
                avarie := "Avarii".avarie_pompa_1,
                mod_selectat := "Simulare_DB".mod_selectat,
                comanda_oprire := "Pompa_DB".comanda_oprire,
                comanda_start := "Pompa_DB".comanda_start,
                feedback => "Pompa_DB".feedback,
                pornire_succes => "Pompa_DB".pornire_succes);
   "Pompa_DB_2"(esd := "Avarii".esd,   // "Pompa"
                avarie := "Avarii".avarie_pompa_auxiliara,
                mod_selectat := "Simulare_DB".mod_selectat,
                comanda_oprire := "Pompa_auxiliara_DB".comanda_oprire,
                comanda_start := "Pompa_auxiliara_DB".comanda_start,
                feedback => "Pompa_auxiliara_DB".feedback,
                pornire_succes => "Pompa_auxiliara_DB".pornire_succes);
END_REGION

REGION Network 11: Simulare
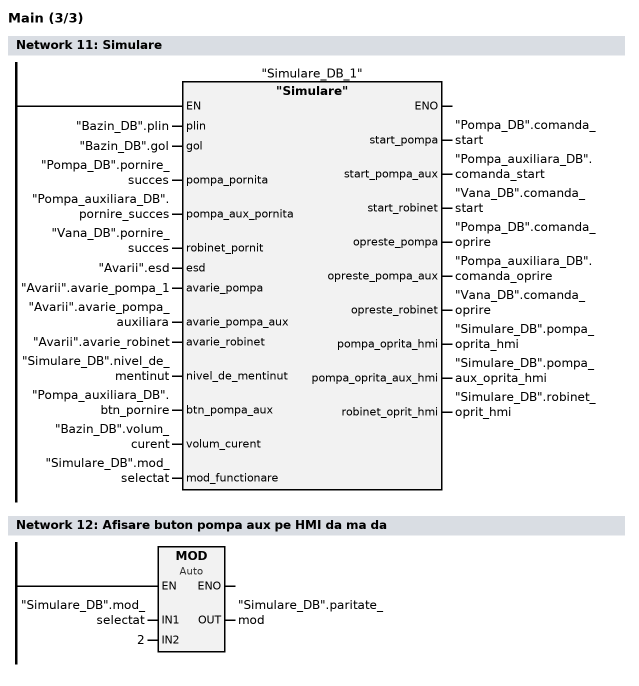
   RUNG wire#powerrail
      "Simulare_DB_1"(plin := "Bazin_DB".plin, gol := "Bazin_DB".gol, pompa_pornita := "Pompa_DB".pornire_succes, pompa_aux_pornita := "Pompa_auxiliara_DB".pornire_succes, robinet_pornit := "Vana_DB".pornire_succes, esd := "Avarii".esd, avarie_pompa := "Avarii".avarie_pompa_1, avarie_pompa_aux := "Avarii".avarie_pompa_auxiliara, avarie_robinet := "Avarii".avarie_robinet, nivel_de_mentinut := "Simulare_DB".nivel_de_mentinut, volum_curent := "Bazin_DB".volum_curent, mod_functionare := "Simulare_DB".mod_selectat, btn_pompa_aux := "Pompa_auxiliara_DB".btn_pornire, start_pompa => "Pompa_DB".comanda_start, start_pompa_aux => "Pompa_auxiliara_DB".comanda_start, start_robinet => "Vana_DB".comanda_start, opreste_pompa => "Pompa_DB".comanda_oprire, opreste_pompa_aux => "Pompa_auxiliara_DB".comanda_oprire, opreste_robinet => "Vana_DB".comanda_oprire, pompa_oprita_hmi => "Simulare_DB".pompa_oprita_hmi, pompa_oprita_aux_hmi => "Simulare_DB".pompa_aux_oprita_hmi, robinet_oprit_hmi => "Simulare_DB".robinet_oprit_hmi)
   END_RUNG
   // the same network as SCL:
   "Simulare_DB_1"(plin := "Bazin_DB".plin,   // "Simulare"
                   gol := "Bazin_DB".gol,
                   pompa_pornita := "Pompa_DB".pornire_succes,
                   pompa_aux_pornita := "Pompa_auxiliara_DB".pornire_succes,
                   robinet_pornit := "Vana_DB".pornire_succes,
                   esd := "Avarii".esd,
                   avarie_pompa := "Avarii".avarie_pompa_1,
                   avarie_pompa_aux := "Avarii".avarie_pompa_auxiliara,
                   avarie_robinet := "Avarii".avarie_robinet,
                   nivel_de_mentinut := "Simulare_DB".nivel_de_mentinut,
                   btn_pompa_aux := "Pompa_auxiliara_DB".btn_pornire,
                   volum_curent := "Bazin_DB".volum_curent,
                   mod_functionare := "Simulare_DB".mod_selectat,
                   start_pompa => "Pompa_DB".comanda_start,
                   start_pompa_aux => "Pompa_auxiliara_DB".comanda_start,
                   start_robinet => "Vana_DB".comanda_start,
                   opreste_pompa => "Pompa_DB".comanda_oprire,
                   opreste_pompa_aux => "Pompa_auxiliara_DB".comanda_oprire,
                   opreste_robinet => "Vana_DB".comanda_oprire,
                   pompa_oprita_hmi => "Simulare_DB".pompa_oprita_hmi,
                   pompa_oprita_aux_hmi => "Simulare_DB".pompa_aux_oprita_hmi,
                   robinet_oprit_hmi => "Simulare_DB".robinet_oprit_hmi);
END_REGION

REGION Network 12: Afisare buton pompa aux pe HMI da ma da
   RUNG wire#powerrail
      Mod(in1 := "Simulare_DB".mod_selectat, in2 := 2, out => "Simulare_DB".paritate_mod)
   END_RUNG
   // the same network as SCL:
   "Simulare_DB".paritate_mod := "Simulare_DB".mod_selectat MOD 2;
END_REGION
END_ORGANIZATION_BLOCK

(* ===== HMI "HMI_RT_1" =====
system functions are stored by id; their names below are inferred from use
connection "HMI_Connection_1": ETHERNET, SMART_S7_1500_OMS

HMI tags "Default tag table"
   "Avarii_esd" : Bool = PLC Avarii.esd, 1 s
   "Avarii_btn_esd" : Bool = PLC Avarii.btn_esd, 1 s
   "Avarii_btn_reset_esd" : Bool = PLC Avarii.btn_reset_esd, 1 s
   "Avarii_avarie_generala" : Bool = PLC Avarii.avarie_generala, 1 s
   "Avarii_avarie_pompa_1" : Bool = PLC Avarii.avarie_pompa_1, 1 s
   "Avarii_avarie_robinet" : Bool = PLC Avarii.avarie_robinet, 1 s
   "Avarii_reset_avarie_generala" : Bool = PLC Avarii.reset_avarie_generala, 1 s
   "Simulare_DB_mod_selectat" : USInt = PLC Simulare_DB.mod_selectat, 1 s
   "Bazin_DB_volum_curent" : Real = PLC Bazin_DB.volum_curent, 1 s
   "Pompa_DB_comanda_oprire" : Bool = PLC Pompa_DB.comanda_oprire, 1 s
   "Pompa_DB_comanda_start" : Bool = PLC Pompa_DB.comanda_start, 1 s
   "Pompa_DB_pornire_succes" : Bool = PLC Pompa_DB.pornire_succes, 1 s
   "Simulare_DB_pompa_oprita_hmi" : Bool = PLC Simulare_DB.pompa_oprita_hmi, 1 s
   "Simulare_DB_robinet_oprit_hmi" : Bool = PLC Simulare_DB.robinet_oprit_hmi, 1 s
   "Robinet_DB_pornit" : Bool = PLC Robinet_DB.pornit, 1 s
   "Alarme_alarme_gather" : Word = PLC Alarme.alarme_gather, 1 s
   "Simulare_DB_nivel_de_mentinut" : Real = PLC Simulare_DB.nivel_de_mentinut, 1 s
   "Vana_DB_pornire_succes" : Bool = PLC Vana_DB.pornire_succes, 1 s
   "Vana_DB_comanda_start" : Bool = PLC Vana_DB.comanda_start, 1 s
   "Pompa_auxiliara_DB_btn_pornire" : Bool = PLC Pompa_auxiliara_DB.btn_pornire, 1 s
   "Simulare_DB_pompa_aux_oprita_hmi" : Bool = PLC Simulare_DB.pompa_aux_oprita_hmi, 1 s
   "Avarii_avarie_pompa_auxiliara" : Bool = PLC Avarii.avarie_pompa_auxiliara, 1 s
   "Pompa_auxiliara_DB_comanda_start" : Bool = PLC Pompa_auxiliara_DB.comanda_start, 1 s
   "Pompa_auxiliara_DB_pornire_succes" : Bool = PLC Pompa_auxiliara_DB.pornire_succes, 1 s
   "Simulare_DB_paritate_mod" : USInt = PLC Simulare_DB.paritate_mod, 1 s

discrete alarms
   1: 'ESD', class Errors, trigger "Alarme_alarme_gather" bit 0
   2: 'Fault at the Pump / Defectiune la pompa', class Errors, trigger "Alarme_alarme_gather" bit 1
   3: 'Fault at the Valve / Defectiune la robinet', class Errors, trigger "Alarme_alarme_gather" bit 2
   4: 'Container full / Bazin plin', class Errors, trigger "Alarme_alarme_gather" bit 3
   5: 'Container empty / Bazin gol', class Errors, trigger "Alarme_alarme_gather" bit 4
   6: 'The required level cannot be 0 / Nivelul cerut nu poate sa fie 0', class Errors, trigger "Alarme_alarme_gather" bit 5
   7: 'Fault at the auxiliar pump / Defectiune la pompa auxiliara', class Errors, trigger "Alarme_alarme_gather" bit 6

text list "Modes": 0 'Empty / Golire'; 1 'Fill / Umplere'; 2 'Auto'

Template "Template_1" 800x480
   Button "Exit" at 722,440 size 55x39; TextOff 'Exit / Iesire'; PictureOff "ExitRuntime_KTP900_Basic_PN_TR"; PictureOn "ExitRuntime_KTP900_Basic_PN_TR"
      on Release: StopRuntime(0)
   Button "Language" at 622,440 size 55x39; TextOff 'Language / Limba'; PictureOff "ToggleLanguage_KTP900_Basic_PN_TR"; PictureOn "ToggleLanguage_KTP900_Basic_PN_TR"
      on Release: function_fb9197e8(-1)
   Button "Start screen" at 520,440 size 55x39; TextOff 'Start screen / Porneste ecranul'; TextOn 'Start screen / Porneste Ecranul'; PictureOff "NavigateHome_KTP900_Basic_PN_TR"; PictureOn "NavigateHome_KTP900_Basic_PN_TR"
      on Release: ActivateScreen("Simulare", 0)

screen "Simulare" 800x480, template "Template_1"
   TextField "Text field_1" at 22,449 size 71x20; Text 'Simulation / Simulare'
   TextField "Text field_2" at 127,449 size 43x20; Text 'Faults / Avarii'
   TextField "Text field_3" at 234,449 size 27x20; Text 'PID'
   TextField "Text field_4" at 323,448 size 51x20; Text 'Alarms / Alarme'
   Circle "Circle_4" at 42,13 size 48x48
      Appearance <- "Avarii_esd"
   Button "Button_4" at 32,72 size 71x32; TextOff 'ESD'
      on Click: SetBit("Avarii_btn_esd")
   Button "Button_5" at 32,115 size 71x32; TextOff 'Reset'
      on Click: SetBit("Avarii_btn_reset_esd")
   Bar "Bar_1" at 222,215 size 374x133; MinimumValue 0; MaximumValue 100
      ProcessValue <- "Bazin_DB_volum_curent"
   GraphicView "Graphic view_1" at 74,210 size 150x143; Picture "Graphic_1"
      Visibility <- "Simulare_DB_pompa_oprita_hmi"
   GraphicView "Graphic view_2" at 74,210 size 150x143; Picture "Graphic_2"
      Visibility <- "Avarii_avarie_pompa_1"
   GraphicView "Graphic view_3" at 74,210 size 150x143; Picture "Graphic_3"
      Visibility <- "Pompa_DB_comanda_start"
   GraphicView "Graphic view_4" at 74,210 size 150x143; Picture "Graphic_4"
      Visibility <- "Pompa_DB_pornire_succes"
   GraphicView "Graphic view_5" at 591,196 size 83x69; Picture "Graphic_10"
      Visibility <- "Simulare_DB_robinet_oprit_hmi"
   GraphicView "Graphic view_6" at 591,195 size 83x69; Picture "Graphic_11"
      Visibility <- "Avarii_avarie_robinet"
   GraphicView "Graphic view_9" at 671,181 size 128x109; Picture "Graphic_14"
      Visibility <- "Simulare_DB_robinet_oprit_hmi"
   IOField "I/O field_1" at 370,169 size 96x32; FormatPattern 999.99; Unit L
      ProcessValue <- "Bazin_DB_volum_curent"
   IOField "I/O field_2" at 353,72 size 71x32; FormatPattern 999.99; Unit L
      Visibility <- "Simulare_DB_mod_selectat"
      ProcessValue <- "Simulare_DB_nivel_de_mentinut"
   SymbolicIOField "Symbolic I/O field_1" at 200,72 size 136x32; TextOff '0'; TextOn '1'; TextList "Modes"
      ProcessValue <- "Simulare_DB_mod_selectat"
   TextField "Text field_5" at 203,46 size 118x20; Text 'Select mode / Selecteaza modul'
   Button "Button_1" at 201,115 size 80x32; TextOff 'Aux Pump / Pompa Aux.'
      on Click: SetBit("Pompa_auxiliara_DB_btn_pornire")
      Visibility <- "Simulare_DB_paritate_mod"
   GraphicView "Graphic view_10" at 406,349 size 96x119; Picture "Graphic_15"
      Visibility <- "Simulare_DB_pompa_aux_oprita_hmi"
   GraphicView "Graphic view_11" at 405,348 size 97x120; Picture "Graphic_16"
      Visibility <- "Avarii_avarie_pompa_auxiliara"
   GraphicView "Graphic view_12" at 404,348 size 98x120; Picture "Graphic_17"
      Visibility <- "Pompa_auxiliara_DB_comanda_start"
   GraphicView "Graphic view_13" at 405,349 size 97x119; Picture "Graphic_18"
      Visibility <- "Pompa_auxiliara_DB_pornire_succes"
   GraphicView "Graphic view_8" at 591,195 size 83x69; Picture "Graphic_13"
      Visibility <- "Vana_DB_comanda_start"
   GraphicView "Graphic view_15" at 670,183 size 130x105; Picture "Graphic_21"
      Visibility <- "Avarii_avarie_robinet"
   GraphicView "Graphic view_7" at 591,195 size 83x69; Picture "Graphic_12"
      Visibility <- "Vana_DB_pornire_succes"
   GraphicView "Graphic view_16" at 670,182 size 130x106; Picture "Graphic_20"
      Visibility <- "Vana_DB_comanda_start"
   GraphicView "Graphic view_14" at 670,182 size 130x108; Picture "Graphic_19"
      Visibility <- "Vana_DB_pornire_succes"

screen "Avarii" 800x480, template "Template_1"
   TextField "Text field_1" at 22,449 size 71x20; Text 'Simulation / Simulare'
   TextField "Text field_2" at 127,449 size 43x20; Text 'Faults / Avarii'
   TextField "Text field_3" at 234,449 size 27x20; Text 'PID'
   TextField "Text field_4" at 323,448 size 50x20; Text 'Alarms / Avarii'
   Circle "Circle_1" at 668,48 size 65x65
      Appearance <- "Avarii_avarie_generala"
   TextField "Text field_5" at 633,16 size 138x25; Text 'General fault / Avarie generala'
   Button "Button_1" at 677,166 size 96x32; TextOff 'Pump / Pompa'
      on Click: SetBit("Avarii_avarie_pompa_1")
   Button "Button_2" at 677,266 size 96x32; TextOff 'Valve / Robinet'
      on Click: SetBit("Avarii_avarie_robinet")
   Button "Button_3" at 651,328 size 96x32; TextOff 'Reset'
      on Click: SetBit("Avarii_reset_avarie_generala")
   Circle "Circle_2" at 618,165 size 34x34
      Appearance <- "Avarii_avarie_pompa_1"
   Circle "Circle_3" at 619,263 size 34x34
      Appearance <- "Avarii_avarie_robinet"
   Circle "Circle_4" at 42,13 size 48x48
      Appearance <- "Avarii_esd"
   Button "Button_4" at 32,72 size 71x32; TextOff 'ESD'
      on Click: SetBit("Avarii_btn_esd")
   Button "Button_5" at 32,115 size 71x32; TextOff 'Reset'
      on Click: SetBit("Avarii_btn_reset_esd")
   Button "Button_6" at 677,214 size 96x32; TextOff 'Pump Aux / Pompa Aux.'
      on Click: SetBit("Avarii_avarie_pompa_auxiliara")
   Circle "Circle_5" at 618,213 size 34x34
      Appearance <- "Avarii_avarie_pompa_auxiliara"

screen "PID (TBA)" 800x480, template "Template_1"
   TextField "Text field_1" at 22,449 size 71x20; Text 'Simulation / Simulare'
   TextField "Text field_2" at 127,449 size 43x20; Text 'Faults / Avarii'
   TextField "Text field_3" at 234,449 size 27x20; Text 'PID'
   TextField "Text field_4" at 323,448 size 51x20; Text 'Alarms / Alarme'
   Circle "Circle_4" at 42,13 size 48x48
      Appearance <- "Avarii_esd"
   Button "Button_4" at 32,72 size 71x32; TextOff 'ESD'
      on Click: SetBit("Avarii_btn_esd")
   Button "Button_5" at 32,115 size 71x32; TextOff 'Reset'
      on Click: SetBit("Avarii_btn_reset_esd")
*)